TYPE ST_ITC_ZoneCommandsEmulation :
(**************************************************************************************
 * 	Application		:	BoxControl Framework
 *	Revision		:	$Revision: 404529 $
 *	Revision date	:	$Date: 2018-04-23 08:21:38 +0200 (Mo., 23 Apr 2018) $
 *	Last changed by	:	$Author: b7bolm $
 *	URL				:	$URL: http://almscdc.swisslog.com/repo/SWPD/Development/BoxControlFramework/20_Release/trunk/01_Software/BCF/BCF/JumpStart/20_Product/11_Emu/12_E_Functions/10_Lib/10_Conv/01_DUTs/ST_ITC_ZoneCommandsEmulation.TcDUT $
 *
 *	Purpose			:	Zone commands
 *
 * ------------------------------------------------------------------------------------
 *	Copyright Swisslog [IP AG], Switzerland. All rights reserved.
 * 
 * ------------------------------------------------------------------------------------
 *	
 * 	Revision History: 
 *
 * 	VERSION			DATE			INITIALS			DESCRIPTION
 *	0.1				01.01.2001		swl					Example
 *
 **************************************************************************************)	
STRUCT
	AddTU 				: BOOL; // Command to add a TU
	RemoveTU			: BOOL; // Command to remove a TU
	Error				: BOOL; // Command to set and reset an error
	TU_DataIndexToAdd 	: DINT; // Index of the TU-Data which has to be added at location -> ADD-TU-Function
	IndexToRemove		: DINT; // TU index to remove 
	ErrorCode			: INT; // ErrorCode for the error which has to be produced
END_STRUCT
END_TYPE

(* stored: Version 1.1.0.1, ProductVersion 3.1.4022.12
   DUT ST_ITC_ZoneCommandsEmulation: Id {8d656747-1dde-432b-913c-3495e143e2f3} *)
